(* IEC 61131-3 sources: RetroPLC_IDE/RetroPLC.Shell/ProjectFiles/POUs/FunctionBlocks, 1 file *)

(* ---- MotorController.st ---- *)
FUNCTION_BLOCK MotorController IMPLEMENTS IMotor
VAR_INPUT
    StartRequest : BOOL;
    StopRequest : BOOL;
END_VAR
VAR_OUTPUT
    IsRunning : BOOL;
END_VAR

METHOD PUBLIC Run
    IsRunning := TRUE;
END_METHOD

IF StopRequest THEN
    IsRunning := FALSE;
ELSIF StartRequest THEN
    IsRunning := TRUE;
END_IF;
END_FUNCTION_BLOCK
